(* CoDeSys 2.3 export: ST_PumpCommands.exp *)

(* Data type in Pump *)
(* єЮЬРЭФл гЯаРТЫХЭШп ЭРбЮбЮЬ *)
TYPE ST_PumpCommands :
STRUCT
    (* ѕбЭЮТЭлХ ЪЮЬРЭФл *)
    xStart : BOOL;
    xStop : BOOL;
    xReset : BOOL;
    
    (* АХЦШЬл *)
    eMode : E_PumpMode;
    xModeChangeRequest : BOOL;
    
    (* ·РФРЭШп *)
    rManualSetpoint : REAL;    (* АгзЭРп гбвРТЪР зРбвЮвл *)
    rAutoSetpoint : REAL;      (* °ТвЮЬРвШзХбЪРп гбвРТЪР *)
END_STRUCT
END_TYPE
